PROGRAM ASSIGN_COLUMN
VAR
	//<Read AMS Net ID>
	fbGetLocalNetID					: FB_GetLocalAmsNetId;
	
	tTimeOut  						: TIME := DEFAULT_ADS_TIMEOUT;
	bBusy      						: BOOL;
    bError     						: BOOL;
    nErrId     						: UDINT;
    AddrString 						: STRING; //T_AmsNetId;
    AddrBytes  						: T_AmsNetIdArr;
	iReadNetIDStep					: INT;
	sColumnName						: STRING;
	
	iColumn							: UINT;
//</Read AMS Net ID>
END_VAR


/////////////////////////////////////////////////////////////////////////////////////////////////////////////////////////////////////////////////////////////////////////////////////////////////
//	State machine
/////////////////////////////////////////////////////////////////////////////////////////////////////////////////////////////////////////////////////////////////////////////////////////////////

//<Read AMS Net ID>
	CASE iReadNetIDStep OF 
		0: (*Idle*)
		
			(*State changed*)
			
			(*Action*)
			
			(*Transition*)
			IF bGetAMSNetID THEN 
				iReadNetIDStep										:= 1; // XXX
			END_IF
			
		1: (*XXX*)
		
			(*State changed*)
			
			(*Action*)
			IsNetIDReadOK											:= FALSE;
			
			fbGetLocalNetID(
				bExecute											:= TRUE , 
				tTimeOut											:= T#3000MS , 
				bBusy												=> bBusy, 
				bError												=> bError, 
				nErrId												=> nErrId, 
				AddrString											=> AddrString, 
				AddrBytes											=> AddrBytes);
			
			(*Transition*)
								
			IF (NOT fbGetLocalNetID.bBusy) THEN
				IF (NOT fbGetLocalNetID.bError) THEN
					IsNetIDReadOK									:= TRUE;
					iReadNetIDStep									:= 2;
				ELSE
					;
				END_IF
			END_IF
			
		2: (**)
		
			(*State changed*)
			
			(*Action*)
			fbGetLocalNetID(	
				bExecute											:= FALSE , 
				tTimeOut											:= T#3000MS , 
				bBusy												=> bBusy, 
				bError												=> bError, 
				nErrId												=> nErrId, 
				AddrString											=> AddrString, 
				AddrBytes											=> AddrBytes);
				
			(*Transition*)
			iReadNetIDStep											:= 3;
			
		3: (**)
		
			(*State changed*)
			
			(*Action*)
			FOR iColumn:= 1 TO NO_OF_COLUMN DO
				IF ARR_AMS_NET_ID[iColumn] = AddrString THEN
					IF bDebugCart AND AddrString = '192.168.1.5.1.1' THEN
						bDebugCart									:= FALSE;
						bDebugStation								:= TRUE;
						Logging.fbDebugLog.M_nLogger(iLogLevel:= Logging.fbDebugLog.P_iLogVerbosity, sSource:= '', sMessage:= '==================================================');		
						Logging.fbDebugLog.M_nLogger(iLogLevel:= Logging.fbDebugLog.P_iLogVerbosity, sSource:= '', sMessage:= CONCAT('AUTO ASIGNED COLUMN NAME ::', 'DEBUG STATION'));			
						Logging.fbDebugLog.M_nLogger(iLogLevel:= Logging.fbDebugLog.P_iLogVerbosity, sSource:= '', sMessage:= '==================================================');
					END_IF
					
					//IF ARR_COL_MOD_ID[iColumn]<> COLUMN_NAME THEN
					//	IsNetIDReadOK := FALSE;
					//END_IF
					COLUMN_NAME										:= ARR_COL_MOD_ID[iColumn];
					IsNetIDReadOK 									:= TRUE;
					iTCColumnID										:=F_GetColumnID(eColumnID:=COLUMN_NAME, sColName=>sColumnName);
					Logging.fbDebugLog.M_nLogger(iLogLevel:= Logging.fbDebugLog.P_iLogVerbosity, sSource:= '', sMessage:= '==================================================');
					Logging.fbDebugLog.M_nLogger(iLogLevel:= Logging.fbDebugLog.P_iLogVerbosity, sSource:= '', sMessage:= CONCAT('Local AMS Net ID ::', AddrString));			
					Logging.fbDebugLog.M_nLogger(iLogLevel:= Logging.fbDebugLog.P_iLogVerbosity, sSource:= '', sMessage:= CONCAT('AUTO ASIGNED COLUMN NAME ::', sColumnName));			
					Logging.fbDebugLog.M_nLogger(iLogLevel:= Logging.fbDebugLog.P_iLogVerbosity, sSource:= '', sMessage:= '==================================================');
        			EXIT;
				ELSE
					IsNetIDReadOK 									:= FALSE;
				END_IF
			END_FOR
			
			IF (NOT IsNetIDReadOK) THEN
				Logging.fbDebugLog.M_nLogger(iLogLevel:= Logging.fbDebugLog.P_iLogVerbosity, sSource:= '', sMessage:= 'XXXXXXXXXXXXXXXXXXXXXXXXXXXXXXXXXXXXXXXXXXXXXXXXXX');
				Logging.fbDebugLog.M_nLogger(iLogLevel:= Logging.fbDebugLog.P_iLogVerbosity, sSource:= '', sMessage:= CONCAT('Invalid Local AMS Net ID ::', AddrString));			
				Logging.fbDebugLog.M_nLogger(iLogLevel:= Logging.fbDebugLog.P_iLogVerbosity, sSource:= '', sMessage:= CONCAT('DEFAULT COLUMN NAME ::', sColumnName));			
				Logging.fbDebugLog.M_nLogger(iLogLevel:= Logging.fbDebugLog.P_iLogVerbosity, sSource:= '', sMessage:= 'XXXXXXXXXXXXXXXXXXXXXXXXXXXXXXXXXXXXXXXXXXXXXXXXXX');
			END_IF
				
			(*Transition*)
			iReadNetIDStep											:= -1; // Only execute get local Net ID one tiime
	END_CASE

//</Read AMS Net ID>

END_PROGRAM

(* stored: Version 1.1.0.1, ProductVersion 3.1.4022.18
   POU ASSIGN_COLUMN: Id {6eb080dd-2815-4167-8240-e347597517d8}, SpecialFunc None *)
